# EPICS substitutions: db/Beckhoff_3XXX/ecmcEL3311.substitutions
file "ecmc_analogInput-chX.template"
{
  pattern {CH_ID, ESLO, EOFF, EGU, PREC}
          {01, "${_ESLO=0.1}", "${_EOFF=0}", "${_EGU=DegC}", "${_PREC=2}"}
}

file "ecmc_status_analog-chX.template"
{
  pattern {CH_ID}
          {01   }
}
